FUNCTION "ST10_Analog" : Void
{ S7_Optimized_Access := 'TRUE' }
VERSION : 0.1
// ATTRIBUTES
// AUTO_NUMBER = False
// BLOCK_NUMBER = 1080
// END_ATTRIBUTES
   VAR_INPUT
      iSysMode : "RCS_SysComInterface_V1";
   END_VAR

   VAR_TEMP
      idex : Int;
   END_VAR


BEGIN


	REGION 氮气压模拟量
	    //定义编号
	    #idex := 1;
	    //功能块调用

	 END_REGION






END_FUNCTION

